// Mitsubishi GX Works2 project: 타이머 예제 1_3   PLC: Q03UDV

PROGRAM MAIN
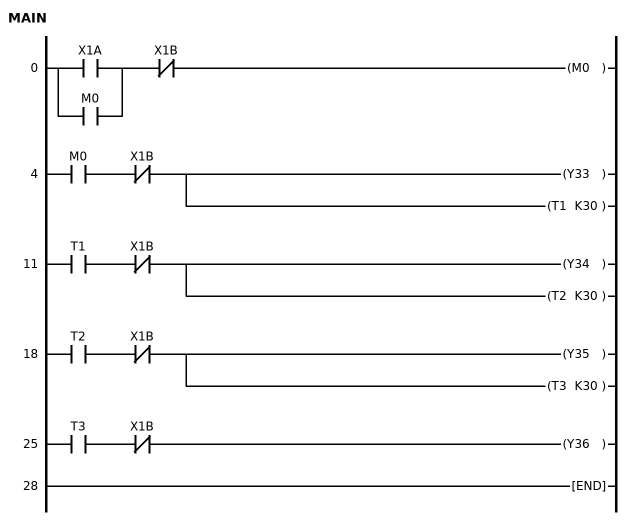
0     LD      X1A
      OR      M0
      ANI     X1B
      OUT     M0
4     LD      M0
      ANI     X1B
      OUT     Y33
      OUT     T1 K30
11    LD      T1
      ANI     X1B
      OUT     Y34
      OUT     T2 K30
18    LD      T2
      ANI     X1B
      OUT     Y35
      OUT     T3 K30
25    LD      T3
      ANI     X1B
      OUT     Y36
28    END
END_PROGRAM
